{region '#Template'}
	{attribute 'Version' := '5.1.0.0'}
	{attribute 'Tags' := '"LCID": "1031", "Text": "Gebäudeautomation, Feueralarm"'}
	{attribute 'Tags' := '"LCID": "1033", "Text": "Building automation, Fire alarm"'}
	{attribute 'Using' := '"Type": "Template", "URI": "Site"'}		 
	{attribute 'Using' := '"Type": "Template", "URI": "EC_ID"'}
	{attribute 'Using' := '"Type": "Template", "URI": "ST_BA_BuildingAlarms"'}
	{attribute 'Description' := '"LCID": "1031", "Text": "Gebäude Feueralarm"'}
	{attribute 'Description' := '"LCID": "1033", "Text": "Building Fire alarm"'}
{endregion}
FUNCTION_BLOCK FB_BA_FireAlarmSystem EXTENDS FB_BA_View
VAR_INPUT CONSTANT
	FireDetector01			: FB_BA_SensorBinary;              
END_VAR	
VAR_OUTPUT
END_VAR

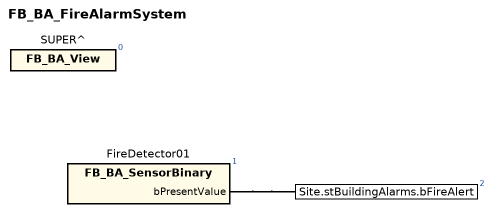
SUPER^(); // FB_BA_View
FireDetector01(); // FB_BA_SensorBinary
Site.stBuildingAlarms.bFireAlert := FireDetector01.bPresentValue;

METHOD FB_init : BOOL
VAR_INPUT
	bInitRetains : BOOL; // if TRUE, the retain variables are initialized (warm start / cold start)
	bInCopyCode : BOOL;  // if TRUE, the instance afterwards gets moved into the copy code (online change)
END_VAR
FireDetector01.iParent					:= THIS^;	
FireDetector01.iLabel					:= LblCtl_FireDetector;
FireDetector01.eDPADMode				:= E_BA_DPADMode.eInclude;
FireDetector01.Input.iLabel				:= LblFun_DangerAlarm;
FireDetector01.Input.sObjectName		:= '{Idx=51}';
FireDetector01.Input.nEventClassID		:= EC_ID.NC10;
FireDetector01.Input.ePolarity			:= E_BA_Polarity.eReverse;
FireDetector01.Input.eEnPlantLock		:= E_BA_LockPriority.eNoLock;
END_METHOD

END_FUNCTION_BLOCK

(* stored: Version 1.1.0.1, ProductVersion 3.1.4024.12
   POU FB_BA_FireAlarmSystem: Id {15e80e22-ee66-4015-9244-c7ef97e708c4}, SpecialFunc None
   Method FB_init: Id {5e4eec7a-a70d-4722-b48c-044a20bb7903} *)
